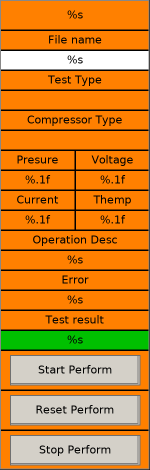
VISUALIZATION vSmallChamber  // 150x470
VAR_IN_OUT
	stParams : stParamsChamber;
	fbChamber : fbChamber;
	stControl : stControl;
END_VAR
    Rectangle (0,390 150x40)
    Rectangle (0,350 150x40)
    Rectangle (0,50 150x20), "%s", text variable: fbChamber.sTestName
        OnMouseClick: write the text variable via VisuDialogs.Keypad
    Rectangle (0,30 150x20), "File name"
    Button (10,355 130x30), "Start Perform", pressed state: stControl.bStartPerform, input disabled if: stControl.bChamberBusy
        OnMouseClick: toggle stControl.bStartPerform
    Rectangle (0,90 150x20), text list: 'txlTestTypes', text index: fbChamber.stControl.iSetTest
    Rectangle (0,70 150x20), "Test Type"
    Rectangle (0,110 150x20), "Compressor Type"
    Rectangle (0,130 150x20), text list: 'txlCompresorTypes', text index: fbChamber.stParams.iCompresorType
    Rectangle (0,150 75x20), "Presure"
    Rectangle (75,150 75x20), "Voltage"
    Rectangle (0,170 75x20), "%.1f", text variable: fbChamber.stInOuts.rPressure
    Rectangle (75,170 75x20), "%.1f", text variable: fbChamber.stInOuts.rVoltage
    Rectangle (0,190 75x20), "Current"
    Rectangle (0,210 75x20), "%.1f", text variable: fbChamber.stInOuts.rVoltage
    Rectangle (0,230 150x20), "Operation Desc"
    Rectangle (0,250 150x20), "%s", text variable: fbChamber.sStepDescription
    Rectangle (0,310 150x20), "Test result"
    Rectangle (0,330 150x20), "%s", text variable: stControl.sTestResult, colour toggle: stControl.sTestResult <> 'DONE'
    Rectangle (0,270 150x20), "Error"
    Rectangle (0,290 150x20), "%s", text variable: stParams.sErrorDescription
    Rectangle (0,0 150x30), "%s", text variable: stParams.sChamberName
    Button (10,395 130x30), "Reset Perform", pressed state: stControl.bResetChamber AND stParams.sErrorDescription = ''
        OnMouseClick: toggle stControl.bResetChamber
    Rectangle (75,190 75x20), "Themp"
    Rectangle (75,210 75x20), "%.1f", text variable: fbChamber.stInOuts.rTemperature
    Rectangle (0,430 150x40)
    Button (10,435 130x30), "Stop Perform", pressed state: stControl.bStopPerform, input disabled if: NOT stControl.bChamberBusy
        OnMouseClick: toggle stControl.bStopPerform
END_VISUALIZATION

(* stored: Version 1.1.0.1, ProductVersion 3.1.4024.12
   Visu vSmallChamber: Id {34be7f7d-21a8-4c05-a62f-26079402c527} *)
